(* PLC project To_FTP_server, Beckhoff Automation GmbH TwinCAT PLC Control 3.5.13.20 *)
(* stored: creationDateTime 2020-09-10T09:40:02.5907467, modificationDateTime 2020-09-10T09:40:02.5907467 *)

FUNCTION_BLOCK FB_LoadDataToWMS
VAR_INPUT
	stLoadIn		:ST_LoadData;
	bEnable			:BOOL;
	iConvStatus		:BYTE;
	bAutomat		:BOOL;
	bMove			:BOOL;
	
END_VAR
VAR_OUTPUT
END_VAR
VAR
	fbStartMove		:R_TRIG;
	fbFinMove		:F_TRIG;
	fbCreateFile: FB_CreateMessage;
	bStartMove:BOOL;
	bEndMove:BOOL;
	fbDelayStartMove:TON;
	fbDelayFinMove:TON;
	bStartSend: BOOL;
	
END_VAR
VAR_IN_OUT
	stLoadMove      :ST_LoadData;
	stLoad			:ST_LoadData;

END_VAR

            fbStartMove(CLK:=bMove);
bStartMove S=fbStartMove.Q;
fbDelayStartMove(IN:=bStartMove,PT:=T#0.3S);
IF bStartMove THEN 
	stLoadMove := stLoadIn;
	IF stLoadMove.sID=stLoadIn.sID  AND  stLoadMove.sWeight=stLoadIn.sWeight OR fbDelayStartMove.Q  THEN
		bStartMove:= FALSE;
	END_IF
END_IF


fbFinMove(CLK:=bMove);
bEndMove S= fbFinMove.Q;
fbDelayFinMove(IN:=bEndMove,PT:=T#0.3S);
IF bEndMove THEN 
	stLoad := stLoadMove;
	IF stLoadMove.sID=stLoad.sID   AND  stLoadMove.sWeight=stLoad.sWeight  OR fbDelayFinMove.Q  THEN
		bEndMove:= FALSE;
	END_IF
END_IF


bStartSend:=bAutomat AND (iConvStatus=2 OR iConvStatus=3) AND NOT bEndMove;
fbCreateFile();
          
END_FUNCTION_BLOCK
